FUNCTION_BLOCK TAdsReadWriteBySymbolName
VAR
    Execution : TExecution;
    StateMonitor : TValueMonitor;
    State : INT;

	AmsNetId : T_AmsNetId;
	Port : T_AmsPort;
	SymbolName : STRING;
    ReadDataAddress : PVOID;
    ReadDataLength : UDINT;
    WriteDataAddress : PVOID;
    WriteDataLength : UDINT;    
    KeepSymbolHandle    : BOOL;  
	SymbolHandle 	   :	DWORD := 0;
    RetryCounter : TCounter;
    
    AdsReadWrite_GetSymHandle : TAdsReadWrite;
    AdsReadWrite_ToSymbol    : TAdsReadWrite;
    AdsWrite_ReleaseSymHandle : TAdsWrite;

END_VAR
VAR CONSTANT
    sInit          : INT := 0;
    sGetHandle     : INT := 1;
    sReadWrite     : INT := 2;
    sReleaseHandle : INT := 3;
END_VAR

StateMonitor.Test(State);
CASE State OF
    sInit:
        IF Execution.Starting THEN
            Execution.SetBusy();
            RetryCounter.Reset();
            IF SymbolHandle = 0 THEN
                State := sGetHandle;
            ELSE
                State := sReadWrite;
            END_IF
		END_IF
        
    sGetHandle:    
        IF StateMonitor.Changed THEN
            // Get a symbol handle from the runtime...
            AdsReadWrite_GetSymHandle.Execute(
                AmsNetId            := AmsNetId, 
                Port                := Port, 
                IndexGroup          := ADSIGRP_SYM_HNDBYNAME, 
                IndexOffset         := 0, 
                ArgsAddress         := ADR(SymbolName), 
                ArgsLength          := INT_TO_UDINT(LEN(SymbolName)), 
                ReturnValueAddress  := ADR(SymbolHandle), 
                ReturnValueLength   := SIZEOF(SymbolHandle));
        ELSE
            IF AdsReadWrite_GetSymHandle.ExecutionResult.Done THEN
                State := sReadWrite;
			END_IF
            IF AdsReadWrite_GetSymHandle.ExecutionResult.Error THEN
                Execution.SetError(AdsReadWrite_GetSymHandle.ExecutionResult.ErrorId);
                SymbolHandle := 0;
                State := sInit;
			END_IF
        END_IF
        
    sReadWrite:  
        IF StateMonitor.Changed THEN
            // Write the data to the symbol...
            AdsReadWrite_ToSymbol.Execute(
                AmsNetId           := AmsNetId, 
                Port               := Port, 
                IndexGroup         := ADSIGRP_SYM_VALBYHND, 
                IndexOffset        := SymbolHandle, 
                ArgsAddress        := WriteDataAddress, 
                ArgsLength         := WriteDataLength, 
                ReturnValueAddress := ReadDataAddress, 
                ReturnValueLength  := ReadDataLength);
            
        ELSE
            IF AdsReadWrite_ToSymbol.ExecutionResult.Done THEN
                IF KeepSymbolHandle THEN
                    Execution.SetDone();
                    State := sInit;
                ELSE
                    State := sReleaseHandle;
				END_IF
                
            ELSIF AdsReadWrite_ToSymbol.ExecutionResult.Error THEN
                // Detect if it failed due to an online change invalidating the symbol handle...
                IF 
                    AdsReadWrite_ToSymbol.ExecutionResult.ErrorId = E_AdsErr.DEVICE_SYMBOLVERSIONINVALID 
                 OR
                    AdsReadWrite_ToSymbol.ExecutionResult.ErrorId = E_AdsErr.DEVICE_SYMBOLNOTACTIVE 
                THEN
                    IF RetryCounter.Value > 0 THEN
                        Execution.SetError(AdsReadWrite_ToSymbol.ExecutionResult.ErrorId);
                        SymbolHandle := 0;
                        State := sInit;
                    ELSE
                        RetryCounter.Inc();
                        SymbolHandle := 0;
                        State := sGetHandle;
                    END_IF
                ELSE
                    State := sReleaseHandle;
				END_IF
			END_IF
		END_IF

    sReleaseHandle:    
        IF StateMonitor.Changed THEN
            // Release the symbol handle......
            AdsWrite_ReleaseSymHandle.Execute(
                AmsNetId        := AmsNetId, 
                Port            := Port, 
                IndexGroup      := ADSIGRP_SYM_RELEASEHND, 
                IndexOffset     := SymbolHandle, 
                DataLength      := 0, 
                DataAddress     := 0);
        ELSE
            IF AdsWrite_ReleaseSymHandle.ExecutionResult.Done THEN
                // Handle write error to the symbol...
                IF AdsReadWrite_ToSymbol.ExecutionResult.Error THEN
                    Execution.SetError(AdsReadWrite_ToSymbol.ExecutionResult.ErrorId);
                ELSE
                    Execution.SetDone();
				END_IF
                SymbolHandle := 0;
                State := sInit;
            ELSIF AdsWrite_ReleaseSymHandle.ExecutionResult.Error THEN
                // Handle release handle error...
                Execution.SetError(AdsWrite_ReleaseSymHandle.ExecutionResult.ErrorId);
                SymbolHandle := 0;
                State := sInit;
			END_IF
		END_IF

END_CASE

AdsReadWrite_GetSymHandle();
AdsReadWrite_ToSymbol();
AdsWrite_ReleaseSymHandle();

METHOD Execute : BOOL
VAR_INPUT
	AmsNetId : T_AmsNetId;
	Port : T_AmsPort;
	SymbolName : STRING;
    ReadDataAddress : PVOID;
    ReadDataLength : UDINT;
    WriteDataAddress : PVOID;
    WriteDataLength : UDINT;
    KeepSymbolHandle    : BOOL;  
END_VAR
THIS^.AmsNetId          := AmsNetId;
THIS^.Port              := Port;
THIS^.SymbolName        := SymbolName;
THIS^.ReadDataAddress   := ReadDataAddress;
THIS^.ReadDataLength    := ReadDataLength;
THIS^.WriteDataAddress  := WriteDataAddress;
THIS^.WriteDataLength   := WriteDataLength;
THIS^.KeepSymbolHandle  := KeepSymbolHandle;

Execute := Execution.Start();
END_METHOD

PROPERTY ExecutionResult : IExecutionResult
GET
ExecutionResult := Execution;
END_GET
END_PROPERTY

END_FUNCTION_BLOCK

(* stored: Version 1.1.0.1, ProductVersion 3.1.4024.3
   POU TAdsReadWriteBySymbolName: Id {13f7dcd6-ccb9-0900-2fd9-3c87339f9e7d}, SpecialFunc None
   Method Execute: Id {8ce67ebf-85ed-4725-8a35-b4f7e3fd3524}
   Property ExecutionResult: Id {4f62956f-a162-0900-311d-9b0770251f12}
   Get Get: Id {5a2dab17-8cca-0dc8-3846-dd0376db8641} *)
